// Gets the lower bound index of the array of specified type.
FUNCTION F_GetXIntArrayLowerBound : T_Position // The lower bound index of the specified array.
VAR_IN_OUT
	arArray : ARRAY[*] OF __XINT; // The array to query.
END_VAR

F_GetXIntArrayLowerBound := LOWER_BOUND(arArray, 1);

END_FUNCTION

(* stored: Version 1.1.0.1
   POU F_GetXIntArrayLowerBound: Id {f7d84ce4-f70e-0ab9-2877-1e33917ff41b}, SpecialFunc None *)
